INTERFACE ITF_Invoerband

PROPERTY Status : PackMLStates
GET
END_GET
END_PROPERTY

METHOD Update : BOOL
VAR_INPUT
END_VAR
END_METHOD

END_INTERFACE

(* stored: Version 1.1.0.1
   Itf ITF_Invoerband: Id {208c2622-9311-49c8-a388-bf23b5f5485c}
   Property Status: Id {cc9c15ef-cfd9-4747-b758-1a77f85a9f4b}
   Get Get: Id {0a476c26-0988-4832-897b-a16c89844ce0}
   Method Update: Id {58b6eaaa-993c-4b51-b9af-3f8615c521ee} *)
